PROGRAM ModbusCommunication
VAR
	aP1, aP2				: ARRAY [GrundfosRegAddress.listStart..GrundfosRegAddress.listEnd] OF WORD;
	aFeeder					: ARRAY [ATV212RegAddress.listStart..ATV212RegAddress.listEnd] OF WORD;
	nStep					: INT := 0;
END_VAR

VAR CONSTANT
	bP1Addr					: BYTE := 2;
	bP2Addr					: BYTE := 4;
	bFeederAddr				: BYTE := 5;
	wStartPumpCmd			: WORD := 16#0000;
	wStopPumpCmd			: WORD := 16#8000;
END_VAR

HWVar.ModbusMaster.ReadRegs(Execute := FALSE);
HWVar.ModbusMaster.WriteRegs(Execute := FALSE);
CASE nStep OF
	0:
		P1Read();
	1:
		P2Read();
	2:
		GrundfosDataConversion(arrReg:= aP1, pstGrundfosMagna3:= ADR(GVL.stP1));
		GrundfosDataConversion(arrReg:= aP2, pstGrundfosMagna3:= ADR(GVL.stP2));
		nStep := 3;
	3:	
		FeederRead();
	4:
		ATV212DataConversion(arrReg:=aFeeder, pstATV212:= ADR(GVL.stFeeder));
		nStep := 0;
END_CASE;

METHOD PRIVATE _P1Read : BOOL
VAR_STAT
	nRegisterAddress	: GrundfosRegAddress;
END_VAR
IF (NOT HWVar.ModbusMaster.BUSY) THEN
	HWVar.ModbusMaster.ReadRegs(
		UnitID := bP1Addr,
		Quantity := 1,
		MBAddr := nRegisterAddress,
		cbLength := 2,
		pMemoryAddr := ADR(aP1[nRegisterAddress]),
		Execute := TRUE,
		Timeout := T#5S,
		BUSY => ,
		Error =>
		);
	nRegisterAddress := nRegisterAddress+1;
	IF (nRegisterAddress = GrundfosRegAddress.listEnd + 1) THEN
		nStep := 1;
		nRegisterAddress :=  GrundfosRegAddress.listStart;
	END_IF
END_IF;
END_METHOD

METHOD PRIVATE _P2Read : BOOL
VAR_STAT
	nRegisterAddress	: GrundfosRegAddress;
END_VAR
IF (NOT HWVar.ModbusMaster.BUSY) THEN
	HWVar.ModbusMaster.ReadRegs(
		UnitID := bP2Addr,
		Quantity := 1,
		MBAddr := nRegisterAddress,
		cbLength := 2,
		pMemoryAddr := ADR((aP2[nRegisterAddress])),
		Execute := TRUE,
		Timeout := T#5S,
		BUSY => ,
		Error =>
		);
	nRegisterAddress := nRegisterAddress+1;
	IF (nRegisterAddress = GrundfosRegAddress.listEnd+1) THEN
		nStep := 2;
		nRegisterAddress :=  GrundfosRegAddress.listStart;
	END_IF
END_IF;
END_METHOD

METHOD ATV212DataConversion : BOOL
VAR_INPUT
	arrReg	: ARRAY [ATV212RegAddress.listStart..ATV212RegAddress.listEnd] OF WORD;
	pstATV212	: POINTER TO ATV212;
END_VAR

VAR
	iMemIndex: ATV212RegAddress;
	iRegIndex: ATV212RegAddress;
	a_MbRegValue	: ARRAY [300..350] OF REAL;
	dwMergedReg		: DWORD;
END_VAR
WHILE (iMemIndex <  ATV212RegAddress.listEnd AND iRegIndex < 879) DO
	IF (iRegIndex <> 875)
		AND (iRegIndex <> 876) 
		AND (iRegIndex <> 877)
		AND (iRegIndex <> 878) THEN
		a_MbRegValue[iRegIndex] := (arrReg[iMemIndex])*Scale.fATV212Scale[iRegIndex];
		iMemIndex := iMemIndex + 1;
		iRegIndex := iRegIndex + 1;
	ELSE
		dwMergedReg := SHL(WORD_TO_DWORD(arrReg[iMemIndex]),16) OR WORD_TO_DWORD(arrReg[iMemIndex+1]);
		a_MbRegValue[iRegIndex] := (dwMergedReg)*Scale.fATV212Scale[iRegIndex];
		iMemIndex := iMemIndex + 2;
		iRegIndex := iRegIndex + 1;
	END_IF
END_WHILE
MEMCPY(pstATV212, ADR(a_MbRegValue), SIZEOF(ATV212));
END_METHOD

METHOD FeederRead : BOOL
VAR_INPUT
END_VAR
IF (NOT HWVar.ModbusMaster.BUSY) THEN
	HWVar.ModbusMaster.ReadRegs(
		UnitID := bFeederAddr,
		Quantity := 4,
		MBAddr := 875,
		cbLength := SIZEOF(aFeeder),
		pMemoryAddr := ADR(aFeeder),
		Execute := TRUE,
		Timeout := T#5S,
		BUSY => ,
		Error =>
		);
		nStep := 4;
END_IF
END_METHOD

METHOD PUBLIC GrundfosDataConversion : BOOL
VAR_INPUT
	arrReg	: ARRAY [GrundfosRegAddress.listStart..GrundfosRegAddress.listEnd] OF WORD;
	pstGrundfosMagna3	: POINTER TO GrundfosMagna3;
END_VAR

VAR
	iMemIndex: GrundfosRegAddress;
	iRegIndex: GrundfosRegAddress;
	a_MbRegValue	: ARRAY [300..350] OF REAL;
	dwMergedReg		: DWORD;
END_VAR
WHILE (iMemIndex <  GrundfosRegAddress.listEnd AND iRegIndex < 351) DO
	IF (iRegIndex <> 311) 
		AND (iRegIndex <> 326)
		AND (iRegIndex <> 328) 
		AND (iRegIndex <> 331)
		AND (iRegIndex <> 323)
		AND (iRegIndex <> 342)
		AND (iRegIndex <> 351)
		AND (iRegIndex <> 353)
		AND (iRegIndex <> 356)
		AND (iRegIndex <> 358)
		AND (iRegIndex <> 360) THEN
		a_MbRegValue[iRegIndex] := (arrReg[iMemIndex])*Scale.fGrundfosScale[iRegIndex];
		iMemIndex := iMemIndex + 1;
		iRegIndex := iRegIndex + 1;
	ELSE
		dwMergedReg := SHL(WORD_TO_DWORD(arrReg[iMemIndex]),16) OR WORD_TO_DWORD(arrReg[iMemIndex+1]);
		a_MbRegValue[iRegIndex] := (dwMergedReg)*Scale.fGrundfosScale[iRegIndex];
		iMemIndex := iMemIndex + 2;
		iRegIndex := iRegIndex + 1;
	END_IF
END_WHILE
MEMCPY(pstGrundfosMagna3, ADR(a_MbRegValue), SIZEOF(GrundfosMagna3));
END_METHOD

METHOD PRIVATE P1Read : BOOL
VAR_STAT
	nRegisterAddress	: GrundfosRegAddress;
END_VAR
IF (NOT HWVar.ModbusMaster.BUSY) THEN
	HWVar.ModbusMaster.ReadRegs(
		UnitID := bP2Addr,
		Quantity := 62,
		MBAddr := 300,
		cbLength := SIZEOF(aP2),
		pMemoryAddr := ADR(aP2),
		Execute := TRUE,
		Timeout := T#5S,
		BUSY => ,
		Error =>
		);
		nStep := 1;
END_IF;
END_METHOD

METHOD PRIVATE P2Read : BOOL
VAR_STAT
	nRegisterAddress	: GrundfosRegAddress;
END_VAR
IF (NOT HWVar.ModbusMaster.BUSY) THEN
	HWVar.ModbusMaster.ReadRegs(
		UnitID := bP1Addr,
		Quantity := 62,
		MBAddr := 300,
		cbLength := SIZEOF(aP1),
		pMemoryAddr := ADR(aP1),
		Execute := TRUE,
		Timeout := T#5S,
		BUSY => ,
		Error =>
		);
		nStep := 2;
END_IF;
END_METHOD

ACTION SC01Read:
nStep := 3;
END_ACTION

END_PROGRAM

(* stored: Version 1.1.0.1, ProductVersion 3.1.4022.18
   POU ModbusCommunication: Id {bf59a4bc-9bbb-44a9-a9e0-c1d2c7fb1f0e}, SpecialFunc None
   Method _P1Read: Id {b9f1af86-d931-4bc8-9247-4c25a97ce7f9}
   Method _P2Read: Id {4de9e116-2209-4dad-8d5a-4715edb7e7e7}
   Method ATV212DataConversion: Id {f7c5cd8b-45b5-444d-bc30-c649d80180e3}
   Method FeederRead: Id {0e093eec-6a04-471a-b96f-3c921f9b1d43}
   Method GrundfosDataConversion: Id {e207b614-c65b-464e-b6c3-2ac0f5daff8e}
   Method P1Read: Id {37f61ac5-bad2-4bc1-a0c5-9c26c5ca0162}
   Method P2Read: Id {335cbb27-56a2-45cb-b675-2b8cdf6cd692}
   Action SC01Read: Id {ec0a3cb0-d056-4f29-9dbb-7c9033aa133f} *)
